(* CODESYS project EZS3_Template.project

Project tree, tasks and I/O mapping:
  Device : Berghof PPC V3 Control, Berghof Automation GmbH, version 3.12.3.0
    application Application
      libraries: Standard, * (System)
      task MainTask (cyclic, interval 4000 µs, priority 0) calls EtherCAT_Master.EtherCAT_Task [EtherCAT_Master.EtherCAT_Task], MAIN
      task EtherCAT_Task (cyclic, interval 4000 µs, priority 0) calls EtherCAT_Master.EtherCAT_Task [EtherCAT_Master.EtherCAT_Task]
      program MAIN [FBD]
      global variables Globale_Variablen
      ControlLogic/
        program Control [ST]
        function block ConveyorStation [FBD]: delivered, deliver, init, initialized, transported, transport, waitForSuccessor
        function block StationSequence [SFC]: Init_active
        function block DeliveryStation [ST]: delivered, initialized, transported, deliver, init, transport, waitForSuccessor
      Interface/
        interface IStation: deliver, init, transport, waitForSuccessor, delivered, initialized, transported
      Simulation/
        function block SimSlider [ST]
        function block SimWerkstueck [SFC]: Init_entry, Band1_active, Schieber1_active, Band2_active, Band3_active, Schieber2_active, Band4_active
        program SimulationPRG [ST]
        program Simu [ST]
      visualisation TAKTSTRASSE
    EtherCAT_Master : EtherCAT Master, 3S - Smart Software Solutions GmbH, version 3.5.8.40
        settings: NetworkName = 'eth1'; NetworkName = "eth1"; SelectNetworkByName = True
      onboard_Buskoppler : onboard Buscoupler, Berghof Automation GmbH, version Revision=16#00000001
          settings: DC sync0 cycletime = 4000; DC sync1 cycletime = 4000
        E_I_O_DI16_DO16 : DI16/DO16 1ms 0.5A (204 800 100), Berghof Automation GmbH, version Revision=16#00000001
            settings: DC sync0 cycletime = 4000; DC sync1 cycletime = 4000
            unmapped channels: DigitalOutput0, DigitalOutput1, DigitalOutput2, DigitalOutput3, DigitalOutput4, DigitalOutput5, DigitalOutput6, DigitalOutput7, DigitalOutput8, DigitalOutput9, DigitalOutput10, DigitalOutput11, DigitalOutput12, DigitalOutput13, DigitalOutput14, DigitalOutput15, DigitalInput0, DigitalInput1, DigitalInput2, DigitalInput3, DigitalInput4, DigitalInput5, DigitalInput6, DigitalInput7, DigitalInput8, DigitalInput9, DigitalInput10, DigitalInput11, DigitalInput12, DigitalInput13, DigitalInput14, DigitalInput15
  libraries: VisuSymbols, 3.5.10.0 (System)
  text list GlobalTextList
*)

// Device/Application/Globale_Variablen
VAR_GLOBAL
	(**** STUDENTEN VARIABLEN ****)

	L1: BOOL;	(* Lichtschranke 1 (Einlegestation) *) 
	L2: BOOL; 	(* Lichtschranke 2 (Einlegestation) *)
	L3: BOOL; 	(* Lichtschranke 3 (Fraeser) *) 
	L4: BOOL;	(* Lichtschranke 4 (Bohrer) *) 
	L5: BOOL; 	(* Lichtschranke 5 (Ausgabestation) *) 
	
	E1: BOOL; 	(* Endanschlag 1 (Uebergabestation 1) *) 
	E2: BOOL; 	(* Endanschlag 2 (Uebergabestation 1) *) 
	E3: BOOL; 	(* Endanschlag 3 (Uebergabestation 2) *) 
	E4: BOOL; 	(* Endanschlag 4 (Uebergabestation 2) *)
	
	B1 AT %QX0.0: BOOL;	(* Foerderband 1 (Einlegestation) *)
	B2 AT %QX0.1: BOOL; (* Foerderband 2 (Fraeser) *) 
	B3 AT %QX0.2: BOOL; (* Foerderband 3 (Bohrer) *) 
	B4 AT %QX0.3: BOOL; (* Foerderband 4 (Ausgabestation) *) 
	
	M1 AT %QX0.5: BOOL; (* Motor 1 (Uebergabestation 1) *)
	M2 AT %QX0.6: BOOL; (* Motor 2 (Fraeser) *)
	M3 AT %QX0.7: BOOL; (* Motor 3 (Bohrer) *)
	M4 AT %QX0.8: BOOL; (* Motor 4 (Uebergabestation 2) *) 
	
	R1 AT %QX0.10: BOOL; (* Relais 1 (Uebergabestation 1) *) 
	R2 AT %QX0.11: BOOL; (* Relais 2 (Uebergabestation 1) *) 
 
	(***** Bedienpult *****) 
	S1: BOOL; (* Taster 1 (Start) *) 
	S2: BOOL; (* Taster 2 (Stopp) *) 
	H1: BOOL; (* Lampe 1 *) 
	
	(**** ENDE STUDENTEN VARIABLEN ****) 
	
	L1_real AT %IX0.0: BOOL; 	(* Lichtschranke 1 (Einlegestation) *)
	L2_real AT %IX0.1: BOOL; 	(* Lichtschranke 2 (Einlegestation) *) 
	L3_real AT %IX0.2: BOOL; 	(* Lichtschranke 3 (Fraeser) *) 
	L4_real AT %IX0.3: BOOL; 	(* Lichtschranke 4 (Bohrer) *) 
	L5_real AT %IX0.4: BOOL; 	(* Lichtschranke 5 (Ausgabestation) *)

	E1_real AT %IX0.6: BOOL; 	(* Endanschlag 1 (Uebergabestation 1) *)
	E2_real AT %IX0.7: BOOL; 	(* Endanschlag 2 (Uebergabestation 1) *)
	E3_real AT %IX0.8: BOOL; 	(* Endanschlag 3 (Uebergabestation 2) *)
	E4_real AT %IX0.9: BOOL; 	(* Endanschlag 4 (Uebergabestation 2) *) 

	SIMULATION: BOOL := TRUE;  

END_VAR

// Device/Application/MAIN
PROGRAM MAIN
VAR
END_VAR

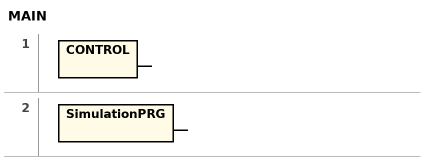
// NETWORK 1
CONTROL();

// NETWORK 2
SimulationPRG();

END_PROGRAM

// Device/Application/ControlLogic/Control
PROGRAM Control
VAR
	input: 		ConveyorStation;
	inputSequence: 		StationSequence; 
	
	deliv1:		DeliveryStation;
	deliv1Seq:	StationSequence;
	active: SR; 
END_VAR

// Initialisation of stations 
//
// Example
// stationXY(inpuX := TRUE, inputY := FALSE); 
// O1 := stationXY.outputV; 
// O2 := stationXY.outputW; 

// Initialisation of function blocks for station sequences 
// 
// Example 
// stationXYSequence(station := stationXY, pieceAvailable := TRUE, nextStationReady := FALSE); 

// Code for the control panel 
active(Set1 := S1, RESET := S2); 
H1 := active.Q1; 

IF active.Q1 THEN 
	
	input(sensorBeltEnd := L2, followUpTime := T#4S);
	B1 := input.beltMotor; 
	inputSequence(station := input, pieceAvailable := L1, nextStationReady :=deliv1.initialized ); 
  	deliv1(start_sensor:=E1,end_sensor:=E2);
	M1:=deliv1.motor;
	R1:=deliv1.relais;
	deliv1Seq(station:=deliv1,pieceAvailable:=input.delivered,nextStationReady:=TRUE);
ELSE 
	// TODO set all motors to stop/pause 
	B1 := FALSE; 
END_IF

END_PROGRAM

// Device/Application/ControlLogic/ConveyorStation
FUNCTION_BLOCK ConveyorStation IMPLEMENTS IStation
VAR_INPUT
	sensorBeltEnd:	BOOL;
	followUpTime: 	TIME; 
END_VAR
VAR_OUTPUT
	beltMotor: BOOL; 
END_VAR
VAR
	followUpTimer: TON; 
END_VAR

PROPERTY delivered : BOOL
GET
delivered := followUpTimer.Q;
END_GET
END_PROPERTY

METHOD deliver
// after followUpTime the deliverDone method should trigger 
followUpTimer(IN := TRUE, PT := followUpTime); 
beltMotor := NOT followUpTimer.Q;
END_METHOD

METHOD init
// reinitialize timer to clear it 
followUpTimer(IN := FALSE, PT := followUpTime); 
beltMotor := FALSE;
END_METHOD

PROPERTY initialized : BOOL
GET
initialized:=(not beltMotor) and (not sensorBeltEnd);
END_GET
END_PROPERTY

PROPERTY transported : BOOL
GET
transported:=sensorBeltEnd;
END_GET
END_PROPERTY

METHOD transport
beltMotor:=TRUE;
END_METHOD

METHOD waitForSuccessor
beltMotor:=FALSE;
END_METHOD

END_FUNCTION_BLOCK

// Device/Application/Interface/IStation
INTERFACE IStation

METHOD deliver
VAR_INPUT
END_VAR
END_METHOD

METHOD init
VAR_INPUT
END_VAR
END_METHOD

METHOD transport
VAR_INPUT
END_VAR
END_METHOD

METHOD waitForSuccessor
VAR_INPUT
END_VAR
END_METHOD

PROPERTY delivered : BOOL
GET
END_GET
END_PROPERTY

PROPERTY initialized : BOOL
GET
END_GET
END_PROPERTY

PROPERTY transported : BOOL
GET
END_GET
END_PROPERTY

END_INTERFACE

// Device/Application/ControlLogic/StationSequence
FUNCTION_BLOCK StationSequence
VAR_INPUT
	station: IStation; 
	pieceAvailable: BOOL; 
	nextStationReady: BOOL; 
END_VAR
VAR_OUTPUT
	pieceDelivered: BOOL := FALSE; 
	stationReady: BOOL := FALSE; 
END_VAR
VAR
END_VAR

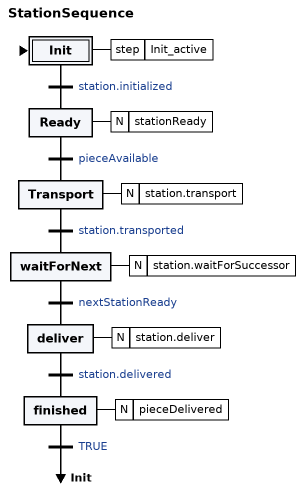
INITIAL_STEP Init:
    Init_active(N);  // step action
END_STEP
TRANSITION FROM Init TO Ready
    := station.initialized;
END_TRANSITION
STEP Ready:
    stationReady(N);
END_STEP
TRANSITION FROM Ready TO Transport
    := pieceAvailable;
END_TRANSITION
STEP Transport:
    station.transport(N);
END_STEP
TRANSITION FROM Transport TO waitForNext
    := station.transported;
END_TRANSITION
STEP waitForNext:
    station.waitForSuccessor(N);
END_STEP
TRANSITION FROM waitForNext TO deliver
    := nextStationReady;
END_TRANSITION
STEP deliver:
    station.deliver(N);
END_STEP
TRANSITION FROM deliver TO finished
    := station.delivered;
END_TRANSITION
STEP finished:
    pieceDelivered(N);
END_STEP
TRANSITION FROM finished TO Init
    := TRUE;
END_TRANSITION

ACTION Init_active:
station.init();
END_ACTION

END_FUNCTION_BLOCK

// Device/Application/ControlLogic/DeliveryStation
FUNCTION_BLOCK DeliveryStation IMPLEMENTS IStation
VAR_INPUT
	start_sensor: BOOL;		(* Wert des ersten Sensors - Schieber ist eingefahren *)
	end_sensor: BOOL;	
	
END_VAR
VAR_OUTPUT
	relais:BOOL;
	motor:BOOL;
END_VAR
VAR
END_VAR


PROPERTY delivered : BOOL
GET
delivered:=end_sensor;
END_GET
END_PROPERTY


PROPERTY initialized : BOOL
GET
initialized:=start_sensor;
END_GET
END_PROPERTY


PROPERTY transported : BOOL
GET
transported:=true;
END_GET
END_PROPERTY

METHOD deliver
relais:=FALSE;
Motor:=True;
END_METHOD


METHOD init
relais:=TRUE;
IF not start_sensor THEN
	motor:=TRUE;
END_IF
END_METHOD


METHOD transport
END_METHOD

METHOD waitForSuccessor
motor:=false;
END_METHOD

END_FUNCTION_BLOCK

// Device/Application/Simulation/SimulationPRG
PROGRAM SimulationPRG
VAR
END_VAR

IF (NOT SIMULATION) THEN 
	// set sensors to inputs if real SPS is used 
	L1 := L1_real; 
	L2 := L2_real; 
	L3 := L3_real; 
	L4 := L4_real; 
	L5 := L5_real; 
	
	E1 := E1_real; 
	E2 := E2_real; 
	E3 := E3_real; 
	E4 := E4_real; 
ELSE 
	Simu(); 
END_IF

END_PROGRAM

// Device/Application/Simulation/Simu
PROGRAM Simu
VAR
	schieber1: SimSlider; 		(* Simulationsbaustein für den ersten Schieber *)
	schieber2: SimSlider; 		(* Simulationsbaustein für den zweiten Schieber *)
	token1: SimWerkstueck; 		(* Simulationsbaustein für das erste Werkstück *)
	token2: SimWerkstueck; 		(* Simulationsbaustein für das zweite Werkstück *)  
END_VAR

(* Aufruf des ersten Schiebers *)
schieber1(start_pos := 0, end_pos := 40, motor := M1, relais := R1);
E1 := schieber1.start_sensor;
E2 := schieber1.end_sensor; 

(* Aufruf des zweiten Schiebers *) 
schieber2(start_pos := 0, end_pos := 40, motor := M4, relais := R2); 
E3 := schieber2.start_sensor;
E4 := schieber2.end_sensor; 

(* Aufruf der Werkstücke *) 
token1(schieber1_pos := schieber1.pos, schieber2_pos := schieber2.pos); 
token2(schieber1_pos := schieber1.pos, schieber2_pos := schieber2.pos); 

(* Zuweisungen für die Lichtschranken *)
L1 := token1.L1_token OR token2.L1_token; 
L2 := token1.L2_token OR token2.L2_token; 
L3 := token1.L3_token OR token2.L3_token; 
L4 := token1.L4_token OR token2.L4_token; 
L5 := token1.L5_token OR token2.L5_token;

END_PROGRAM

// Device/Application/Simulation/SimSlider
FUNCTION_BLOCK SimSlider
VAR_INPUT
	start_pos: INT; 	(* Position, wenn der Schieber eingefahren ist *)
	end_pos: INT; 		(* Position, wenn der Schieber ausgefahren ist *)
	motor: BOOL; 		(* Motor des Schiebers *)
	relais: BOOL; 		(* Relais des Schiebers *)
END_VAR
VAR_OUTPUT
	pos: INT := start_pos;	(* Aktuelle Position des Schiebers *) 
	start_sensor: BOOL; 	(* Wert des ersten Sensors (Schieber ist eingefahren) *) 
	end_sensor: BOOL; 		(* Wert des zweiten Sensors (Schieber ist ausgefahren) *)
END_VAR
VAR
END_VAR

start_sensor := (pos = start_pos); 
end_sensor := (pos = end_pos); 

IF (motor) THEN 
	IF (relais AND pos > start_pos) THEN 
		pos := pos - 1; 
	ELSIF (NOT relais AND pos < end_pos) THEN 
		pos := pos + 1; 
	END_IF 	
END_IF

END_FUNCTION_BLOCK

// Device/Application/Simulation/SimWerkstueck
FUNCTION_BLOCK SimWerkstueck
VAR_INPUT
	start: BOOL := FALSE; 		(* Wird von der Visualisierung gesetzt, wenn das Werkstück auf das Band gelegt wird *) 
	schieber1_pos: INT; 		(* Aktuelle Position des ersten Schiebers *)
	schieber2_pos: INT; 		(* Aktuelle Position des zweiten Schiebers *) 
END_VAR
VAR_OUTPUT
	pos_x: INT; 				(* X Position des Werkstücks relativ zum Startpunkt *)
	pos_y: INT; 				(* Y Position des Werkstücks relativ zum Startpunkt *)
	visible: BOOL;				(* True, falls das Werkstück in der Anlage ist *) 
	L1_token: BOOL; 			(* True, falls das Werkstück vor der 1. Lichtschranke ist *)
	L2_token: BOOL; 			(* True, falls das Werkstück vor der 2. Lichtschranke ist *) 
	L3_token: BOOL; 			(* True, falls das Werkstück vor der 3. Lichtschranke ist *) 
	L4_token: BOOL; 			(* True, falls das Werkstück vor der 4. Lichtschranke ist *) 
	L5_token: BOOL; 			(* True, falls das Werkstück vor der 5. Lichtschranke ist *) 
END_VAR
VAR
END_VAR

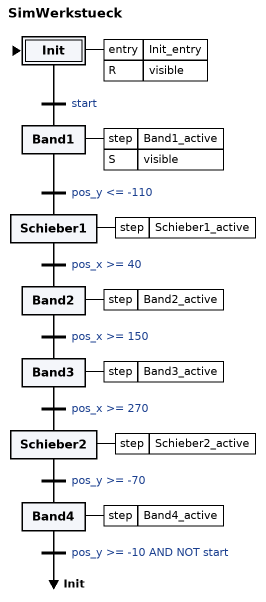
INITIAL_STEP Init:
    Init_entry(P1);  // entry action
    visible(R);
END_STEP
TRANSITION FROM Init TO Band1
    := start;
END_TRANSITION
STEP Band1:
    Band1_active(N);  // step action
    visible(S);
END_STEP
TRANSITION FROM Band1 TO Schieber1
    := pos_y <= -110;
END_TRANSITION
STEP Schieber1:
    Schieber1_active(N);  // step action
END_STEP
TRANSITION FROM Schieber1 TO Band2
    := pos_x >= 40;
END_TRANSITION
STEP Band2:
    Band2_active(N);  // step action
END_STEP
TRANSITION FROM Band2 TO Band3
    := pos_x >= 150;
END_TRANSITION
STEP Band3:
    Band3_active(N);  // step action
END_STEP
TRANSITION FROM Band3 TO Schieber2
    := pos_x >= 270;
END_TRANSITION
STEP Schieber2:
    Schieber2_active(N);  // step action
END_STEP
TRANSITION FROM Schieber2 TO Band4
    := pos_y >= -70;
END_TRANSITION
STEP Band4:
    Band4_active(N);  // step action
END_STEP
TRANSITION FROM Band4 TO Init
    := pos_y >= -10 AND NOT start;
END_TRANSITION

ACTION Init_entry:
pos_x := 0; 
pos_y := 0; 
visible := FALSE; 
L1_token := FALSE; 
L2_token := FALSE; 
L3_token := FALSE; 
L4_token := FALSE; 
L5_token := FALSE;
END_ACTION

ACTION Band1_active:
IF (B1) THEN 
	pos_y := pos_y - 1; 
END_IF

L1_token := (pos_y >= -10); 
L2_token := (pos_y <= -50 AND pos_y >= -70);
END_ACTION

ACTION Schieber1_active:
pos_x := schieber1_pos;
END_ACTION

ACTION Band2_active:
IF (B2) THEN 
	pos_x := pos_x + 1; 
END_IF

L3_token := (pos_x >= 90 AND pos_x <= 110);
END_ACTION

ACTION Band3_active:
IF (B3) THEN 
	pos_x := pos_x + 1; 
END_IF

L4_token := (pos_x >= 200 AND pos_x <= 220);
END_ACTION

ACTION Schieber2_active:
pos_y := -110 + schieber2_pos;
END_ACTION

ACTION Band4_active:
IF (B4) THEN 
	pos_y := pos_y + 1; 
END_IF

L5_token := (pos_y >= -10 AND pos_y <= 10);
END_ACTION

END_FUNCTION_BLOCK

// Device/Application/TAKTSTRASSE
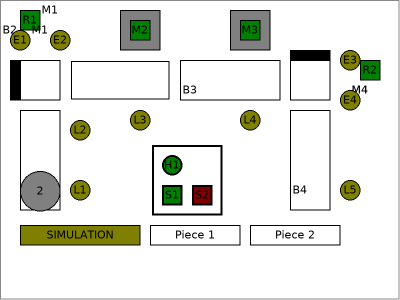
VISUALIZATION TAKTSTRASSE  // 400x300
    Rectangle (20,110 40x100)
    Rectangle (290,60 40x40)
    Rectangle (20,60 40x40)
    RoundedRectangle (20,10 20x20), "R1", colour toggle: Globale_Variablen.R1, input disabled if: (NOT SIMULATION) <> 0
        toggle Globale_Variablen.R1
    RoundedRectangle (360,60 20x20), "R2", colour toggle: R2, input disabled if: NOT SIMULATION
        toggle R2
    RoundedRectangle (150,225 90x20), "Piece 1", colour toggle: Simu.token1.visible, invisible if: NOT SIMULATION
        toggle Simu.token1.start
    RoundedRectangle (20,225 120x20), "SIMULATION", colour toggle: Globale_Variablen.SIMULATION
        toggle Globale_Variablen.SIMULATION
    Polygon (40,30), "M1", colour toggle: Globale_Variablen.M1, invisible if: Globale_Variablen.R1, input disabled if: (NOT SIMULATION) <> 0
        toggle Globale_Variablen.M1
    Polygon (50,10), "M1", colour toggle: Globale_Variablen.M1, invisible if: (NOT R1) <> 0, input disabled if: (NOT SIMULATION) <> 0
        toggle Globale_Variablen.M1
    Polygon (360,90), "M4", colour toggle: M4, invisible if: R2, input disabled if: NOT SIMULATION
        toggle M4
    Polygon (360,90), "M4", colour toggle: M4, invisible if: NOT R2, input disabled if: NOT SIMULATION
        toggle M4
    Rectangle (71,61 98x38)
    Polygon (10,30), "B2", colour toggle: B2, input disabled if: NOT SIMULATION
        toggle B2
    Rectangle (180,60 100x40)
    Polygon (190,90), "B3", colour toggle: B3, input disabled if: NOT SIMULATION
        toggle B3
    Ellipse (130,110 20x20), "L3", colour toggle: L3, input disabled if: NOT SIMULATION
        toggle L3
    Polyline (140,50)
    Ellipse (240,110 20x20), "L4", colour toggle: L4, input disabled if: NOT SIMULATION
        toggle L4
    Polyline (250,50)
    Ellipse (10,30 20x20), "E1", colour toggle: E1, input disabled if: NOT SIMULATION
        toggle E1
    Polygon (30,50)
    Ellipse (50,30 20x20), "E2", colour toggle: E2, input disabled if: NOT SIMULATION
        toggle E2
    Polygon (70,50)
    RoundedRectangle (120,10 40x40)
    RoundedRectangle (130,20 20x20), "M2", colour toggle: M2, input disabled if: NOT SIMULATION
        toggle M2
    RoundedRectangle (230,10 40x40)
    RoundedRectangle (240,20 20x20), "M3", colour toggle: M3, input disabled if: NOT SIMULATION
        toggle M3
    Ellipse (340,50 20x20), "E3", colour toggle: E3, input disabled if: NOT SIMULATION
        toggle E3
    Polygon (340,70)
    Ellipse (340,90 20x20), "E4", colour toggle: E4, input disabled if: NOT SIMULATION
        toggle E4
    Polygon (340,110)
    Ellipse (340,180 20x20), "L5", colour toggle: L5, input disabled if: NOT SIMULATION
        toggle L5
    Ellipse (70,180 20x20), "L1", colour toggle: L1, input disabled if: NOT SIMULATION
        toggle L1
    Polygon (50,200), "B1", colour toggle: B1, input disabled if: NOT SIMULATION
        toggle B1
    Polyline (70,190)
    Ellipse (70,120 20x20), "L2", colour toggle: L2, input disabled if: NOT SIMULATION
        toggle L2
    Polyline (70,130)
    Rectangle (290,110 40x100)
    Polygon (300,190), "B4", colour toggle: B4, input disabled if: NOT SIMULATION
        toggle B4
    Polyline (340,190)
    Ellipse (20,171 40x40), "1", invisible if: NOT Simu.token1.visible
        p3560616238: Simu.token1.pos_x
        p2738717112: Simu.token1.pos_y
    Rectangle (10,60 10x40)
        p3560616238: Simu.schieber1.pos
    Rectangle (290,50 40x10)
        p2738717112: Simu.schieber2.pos
    RoundedRectangle (250,225 90x20), "Piece 2", colour toggle: Simu.token2.visible, invisible if: NOT SIMULATION
        toggle Simu.token2.start
    Ellipse (20,171 40x40), "2", invisible if: NOT Simu.token2.visible
        p3560616238: Simu.token2.pos_x
        p2738717112: Simu.token2.pos_y
    RoundedRectangle (152,145 70x70)
    Ellipse (162,155 20x20), "H1", colour toggle: Globale_Variablen.H1
    RoundedRectangle (162,185 20x20), "S1", colour toggle: Globale_Variablen.S1
        tap Globale_Variablen.S1
    RoundedRectangle (192,185 20x20), "S2", colour toggle: Globale_Variablen.S2
        tap Globale_Variablen.S2
END_VISUALIZATION
